// TIA Portal V17 export
// export: Created 2026-04-13T11:12:41.8804656Z, ExportSetting WithDefaults, DisplayName Totally Integrated Automation Portal, DisplayVersion V17 Update 4, DisplayName TIA Portal Openness, DisplayVersion V17 Update 4, DisplayName TIA Portal Version Control Interface, DisplayVersion V17, DisplayName SINAMICS Startdrive Advanced, DisplayVersion V17, DisplayName SINAMICS Startdrive G130, G150, S120, S150, SINAMICS MV, S210, DisplayVersion V17, DisplayName SINAMICS Startdrive G110M, G120, G120C, G120D, G120P, G115D, DisplayVersion V17, DisplayName STEP 7 Professional, DisplayVersion V17 Update 4, DisplayName STEP 7 Safety, DisplayVersion V17, DisplayName WinCC Professional, DisplayVersion V17 Update 4
FUNCTION_BLOCK "四参数辅助"   // FB42, SCL
{ S7_Optimized_Access := 'TRUE' }
VERSION : 0.1
// stored: AutoNumber true, IsIECCheckEnabled false, IsRetainMemResEnabled false, MemoryReserve 100, SetENOAutomatically false, UDAEnableTagReadback false
   VAR_INPUT
      启动送风机 : Bool;   // 启动送风机命令
      关闭送风机 : Bool;   // 关闭送风机命令
      设定送风流量 : Real;   // 送风流量设定值
      实际送风流量 : Real;   // 流量变送器测量的实际流量
      流量上阈值 : Real := 10.0;   // 合格区间上限偏差值
      流量下阈值 : Real := 5.0;   // 合格区间下限偏差值
   END_VAR
   VAR_IN_OUT
      调节单元 : Real := 4.0;   // 频率调节单元 4Hz/时间
      调节时间 : Real := 30.0;   // 时间为秒
      调节时间PV : Real;
      变频器频率设定 : Real;   // 输出到变频器的频率设定
   END_VAR
   VAR
      运行状态 : Int := 0;   // 0: 停止, 1: 启动中, 2: 运行中, 3: 关闭中
      起始频率 : Real := 10.0;   // 起始频率10Hz
      最高频率 : Real := 50.0;   // 最高频率50Hz
      频率设定值 : Real := 0.0;   // 内部频率设定值
      流量合格 : Bool := FALSE;   // 流量是否在合格区间内
      TON1 : TON_TIME;
   END_VAR
BEGIN

       // 判断流量是否在合格区间内
       #流量合格 := (#实际送风流量 >= (#设定送风流量 - #流量下阈值)) AND
       (#实际送风流量 <= (#设定送风流量 + #流量上阈值));

       // 状态机
       CASE #运行状态 OF
           0:  // 停止状态
               IF #启动送风机 THEN
                   #运行状态 := 1;  // 转到启动状态
                   #频率设定值 := #起始频率;
                  // #送风机运行 := TRUE;
               END_IF;

           1:  // 启动状态
               IF #关闭送风机 THEN
                   #运行状态 := 3;  // 收到关闭命令，转到关闭状态
               ELSIF #流量合格 THEN
                   #运行状态 := 2;  // 流量达到合格区间，转到运行状态
               ELSIF #TON1.Q THEN
                   // 每分钟调整，最多增减4Hz
                   IF #实际送风流量 < #设定送风流量 - #流量下阈值 THEN
                       // 流量不足，增加频率
                       #频率设定值 := #频率设定值 + #调节单元;
                       IF #频率设定值 > #最高频率 THEN
                           #频率设定值 := #最高频率;
                       END_IF;
                   ELSIF #实际送风流量 > #设定送风流量 + #流量上阈值 THEN
                       // 流量过大，减少频率
                       #频率设定值 := #频率设定值 - #调节单元;
                       IF #频率设定值 < #起始频率 THEN
                           #频率设定值 := #起始频率;
                       END_IF;
                   END_IF;
               END_IF;

           2:  // 运行状态（流量稳定）
               IF #关闭送风机 THEN
                   #运行状态 := 3;  // 收到关闭命令，转到关闭状态
               ELSIF NOT #流量合格 AND #TON1.Q THEN
                   #运行状态 := 1;  // 流量不再合格，转回启动状态继续调节
               END_IF;

           3:  // 关闭状态
               IF #TON1.Q THEN
                   // 每分钟减少4Hz
                   #频率设定值 := #频率设定值 - #调节单元;

                   // 频率低于10Hz时关闭送风机
                   IF #频率设定值 < #起始频率 THEN
                     //  #送风机运行 := FALSE;
                       #频率设定值 := #起始频率;
                       #运行状态 := 0;  // 回到停止状态
                   END_IF;
               END_IF;
       END_CASE;

       #TON1(IN:=NOT #TON1.Q,
             PT:=DINT_TO_TIME(REAL_TO_DINT(#调节时间*1000)));

       #调节时间PV:=DINT_TO_REAL(TIME_TO_DINT(#TON1.ET))*1000;
       // 输出频率设定值
       #变频器频率设定 := #频率设定值;
END_FUNCTION_BLOCK
